VISUALIZATION Conveyance  // 2x2
END_VISUALIZATION

(* stored: Version 1.1.0.1, ProductVersion 3.1.4024.15
   Visu Conveyance: Id {7176d18d-8913-488e-836d-46c3f56a0478} *)
